TYPE ST_ITC_IPR :
(**************************************************************************************
 * 	Application		:	BoxControl Framework
 *	Revision		:	$Revision: 404529 $
 *	Revision date	:	$Date: 2018-04-23 08:21:38 +0200 (Mo., 23 Apr 2018) $
 *	Last changed by	:	$Author: b7bolm $
 *	URL				:	$URL: http://almscdc.swisslog.com/repo/SWPD/Development/BoxControlFramework/20_Release/trunk/01_Software/BCF/BCF/JumpStart/20_Product/10_App/11_Com/10_Lib/10_Conv/11_ITC/01_DUTs/ST_ITC_IPR.TcDUT $
 *
 *	Purpose			:	IPR Structure
 *
 * ------------------------------------------------------------------------------------
 *	Copyright Swisslog [IP AG], Switzerland. All rights reserved.
 * 
 * ------------------------------------------------------------------------------------
 *	
 * 	Revision History: 
 *
 * 	VERSION			DATE			INITIALS			DESCRIPTION
 *	0.1				01.01.2001		swl					Example
 *
 **************************************************************************************)
STRUCT
	Position 			: STRING(Conveyor.POSITION_STRINGLENGTH); // 12 Digit SIS Location MM-GGG-EEEE-LLL 
	TU_DataIndex		: DINT; // TU-DataIndex
	MSG_Sequence		: INT; // Assignment message sequence
	TU_ID				: STRING(Conveyor.TU_ID_STRINGLENGTH); // 18 Char SSID
	TU_Type				: INT; // TU-Type
	AssignmentID		: UDINT; // Assignment id
	Height				: INT; // Height Result
	WidthRight			: INT; // Width Right Result
	WidthLeft			: INT; // Width Left Result
	LengthFront			: INT; // Length Front Result
	LengthRear			: INT; // Length Rear Result
	Weight				: DINT; // Weight Value
	Tunnel				: INT; // Tunnel Result
	Runner				: INT; // Runner Result
	ErrorCode			: INT; // Error
	ValidLabelString	: INT; // Valid Label Return Code
	Label				: STRING(Conveyor.LABEL_LENGTH); // Characters of Label Data
END_STRUCT
END_TYPE

(* stored: Version 1.1.0.1, ProductVersion 3.1.4022.12
   DUT ST_ITC_IPR: Id {1737b3f8-a021-4f28-a171-793415da84d2} *)
